TYPE ST_ReloadRoundBelt_Ctrl EXTENDS ST_CommandBasic :
STRUCT
END_STRUCT
END_TYPE

(* stored: Version 1.1.0.1, ProductVersion 3.1.4024.13
   DUT ST_ReloadRoundBelt_Ctrl: Id {2bdf9cc0-b5cb-4421-983e-b5f16d3bf52e} *)
